{attribute addProperty BoxType "EP1312-0001-0016"}
{attribute addProperty Id "A_0038_EP1518_0002_0016EP1518_7C3C20DE36846A_0039_EP1518_0002_0017EP1518_7C3C20DE36846A_0040_EP1518_0002_0018EP1518_7C3C20DE36846A_0041_EP1518_0002_0019EP1518_7C3C20DE36846A_0042_EP1809_0021_0016EP1809_8059E62316020A_0043_EP1809_0021_0017EP1809_8059E62316020A_0044_EP1809_0022_0017EP1809_8059E62316020A_0045_EP1809_0022_0018EP1809_8059E62316020A_0046_EP1809_0042_0018EP1809_FA80E4F816020A_0047_EP1809_0042_0019EP1809_50065817429496726434359738364A_0048_EP1816_0003_0016EP1816_9D1B0E2325632A_0049_EP1816_0008_0016EP1816_D737114C24030A_0050_EP1816_0008_0017EP1816_D737114C24030A_0051_EP1816_0008_0018EP1816_8EE49DA824030A_0052_EP1816_0008_0019EP1816_8EE49DA824030A_0053_EP1816_0008_0020EP1816_8EE49DA824030A_0054_EP1816_1008_0016EP1816_7BF0AF8625632A_0055_EP1816_1008_0017EP1816_7BF0AF8625632A_0056_EP1816_3008_0016EP1816_5F09590E44856A_0057_EP1816_3008_0017EP1816_5F09590E44856A_0058_EP1816_3008_0018EP1816_5F09590E44856A_0059_EP1819_0021_0016EP1819_8059E62316020A_0060_EP1819_0021_0017EP1819_8059E62316020A_0061_EP1819_0022_0016EP1819_8059E62316020A_0062_EP1819_0022_0017EP1819_8059E62316020A_0063_EP1859_0042_0018EP1859_BE389A0216020A_0064_EP1859_0042_0019EP1859_1AE54674429496726434359738364"}
{attribute addProperty CRC "4105665208"}
{attribute addProperty SizeInBites "6320"}
{attribute addProperty SizeInBytes "68719477526"}
TYPE A_0037_EP1312_0001_0016_F4B77AB8 EXTENDS EP1312_179A0949 :
STRUCT
	{attribute addProperty Name "A_0038_EP1518_0002_0016"}
	A_0038_EP1518_0002_0016 : EP1518_7C3C20DE;
	{attribute addProperty Name "A_0039_EP1518_0002_0017"}
	A_0039_EP1518_0002_0017 : EP1518_7C3C20DE;
	{attribute addProperty Name "A_0040_EP1518_0002_0018"}
	A_0040_EP1518_0002_0018 : EP1518_7C3C20DE;
	{attribute addProperty Name "A_0041_EP1518_0002_0019"}
	A_0041_EP1518_0002_0019 : EP1518_7C3C20DE;
	{attribute addProperty Name "A_0042_EP1809_0021_0016"}
	A_0042_EP1809_0021_0016 : EP1809_8059E623;
	{attribute addProperty Name "A_0043_EP1809_0021_0017"}
	A_0043_EP1809_0021_0017 : EP1809_8059E623;
	{attribute addProperty Name "A_0044_EP1809_0022_0017"}
	A_0044_EP1809_0022_0017 : EP1809_8059E623;
	{attribute addProperty Name "A_0045_EP1809_0022_0018"}
	A_0045_EP1809_0022_0018 : EP1809_8059E623;
	{attribute addProperty Name "A_0046_EP1809_0042_0018"}
	A_0046_EP1809_0042_0018 : EP1809_FA80E4F8;
	{attribute addProperty Name "A_0047_EP1809_0042_0019"}
	A_0047_EP1809_0042_0019 : EP1809_50065817;
	{attribute addProperty Name "A_0048_EP1816_0003_0016"}
	A_0048_EP1816_0003_0016 : EP1816_9D1B0E23;
	{attribute addProperty Name "A_0049_EP1816_0008_0016"}
	A_0049_EP1816_0008_0016 : EP1816_D737114C;
	{attribute addProperty Name "A_0050_EP1816_0008_0017"}
	A_0050_EP1816_0008_0017 : EP1816_D737114C;
	{attribute addProperty Name "A_0051_EP1816_0008_0018"}
	A_0051_EP1816_0008_0018 : EP1816_8EE49DA8;
	{attribute addProperty Name "A_0052_EP1816_0008_0019"}
	A_0052_EP1816_0008_0019 : EP1816_8EE49DA8;
	{attribute addProperty Name "A_0053_EP1816_0008_0020"}
	A_0053_EP1816_0008_0020 : EP1816_8EE49DA8;
	{attribute addProperty Name "A_0054_EP1816_1008_0016"}
	A_0054_EP1816_1008_0016 : EP1816_7BF0AF86;
	{attribute addProperty Name "A_0055_EP1816_1008_0017"}
	A_0055_EP1816_1008_0017 : EP1816_7BF0AF86;
	{attribute addProperty Name "A_0056_EP1816_3008_0016"}
	A_0056_EP1816_3008_0016 : EP1816_5F09590E;
	{attribute addProperty Name "A_0057_EP1816_3008_0017"}
	A_0057_EP1816_3008_0017 : EP1816_5F09590E;
	{attribute addProperty Name "A_0058_EP1816_3008_0018"}
	A_0058_EP1816_3008_0018 : EP1816_5F09590E;
	{attribute addProperty Name "A_0059_EP1819_0021_0016"}
	A_0059_EP1819_0021_0016 : EP1819_8059E623;
	{attribute addProperty Name "A_0060_EP1819_0021_0017"}
	A_0060_EP1819_0021_0017 : EP1819_8059E623;
	{attribute addProperty Name "A_0061_EP1819_0022_0016"}
	A_0061_EP1819_0022_0016 : EP1819_8059E623;
	{attribute addProperty Name "A_0062_EP1819_0022_0017"}
	A_0062_EP1819_0022_0017 : EP1819_8059E623;
	{attribute addProperty Name "A_0063_EP1859_0042_0018"}
	A_0063_EP1859_0042_0018 : EP1859_BE389A02;
	{attribute addProperty Name "A_0064_EP1859_0042_0019"}
	A_0064_EP1859_0042_0019 : EP1859_1AE54674;
END_STRUCT
END_TYPE

(* stored: Version 1.2.0.0, ProductVersion 3.1.4024.9
   DUT A_0037_EP1312_0001_0016_F4B77AB8: Id {c933ff0b-1ab2-499f-8997-e01b12f2629c} *)
